// TIA Portal V20 export
DATA_BLOCK "ManualOperationControl_CITIEm1"   // DB447
// stored: MemoryReserve 100
   VAR
      manualOperationEm { ExternalAccessible := 'False'; ExternalVisible := 'False'; ExternalWritable := 'False'} : "LAF_typeManEm";
      manualOperationEmArea { ExternalAccessible := 'False'; ExternalVisible := 'False'; ExternalWritable := 'False'} : Array[1..5] of "LAF_typeManOperationArea";
      manualOperationCms { ExternalAccessible := 'False'; ExternalVisible := 'False'; ExternalWritable := 'False'} : Array[1..41] of "LAF_typeManOperation";
   END_VAR
BEGIN
   manualOperationEm.equipmentModuleNum := 1080;
END_DATA_BLOCK
